{attribute 'qualified_only'}
VAR_GLOBAL
	
	// Heater outputs
	O_HeaterT AT %Q*:BOOL;
	O_HeaterB AT %Q*:BOOL;
	
	// RTD Sensors (PT100)
	I_TermT AT %I*:LREAL;
	I_TermB AT %I*:LREAL;
	
END_VAR

(* stored: Version 1.1.0.1, ProductVersion 3.1.4024.9
   GVL IO: Id {f19c6e7d-dfbd-4478-b507-c13927482bf7} *)
